// Mitsubishi GX Works2 project: q02 최종   PLC: Q02/Q02H

PROGRAM MAIN
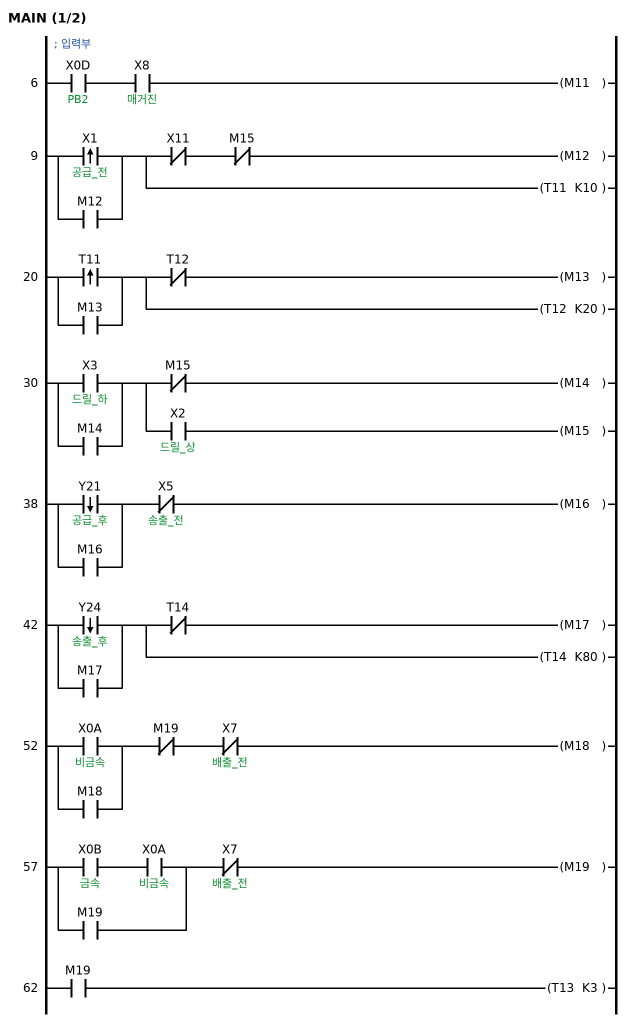
; 입력부
6     LD      X0D  ; PB2
      AND     X8  ; 매거진
      OUT     M11
9     LDP     X1  ; 공급_전
      OR      M12
      MPS
      ANI     X11
      ANI     M15
      OUT     M12
      MPP
      OUT     T11 K10
20    LDP     T11
      OR      M13
      MPS
      ANI     T12
      OUT     M13
      MPP
      OUT     T12 K20
30    LD      X3  ; 드릴_하
      OR      M14
      MPS
      ANI     M15
      OUT     M14
      MPP
      AND     X2  ; 드릴_상
      OUT     M15
38    LDF     Y21  ; 공급_후
      OR      M16
      ANI     X5  ; 송출_전
      OUT     M16
42    LDF     Y24  ; 송출_후
      OR      M17
      MPS
      ANI     T14
      OUT     M17
      MPP
      OUT     T14 K80
52    LD      X0A  ; 비금속
      OR      M18
      ANI     M19
      ANI     X7  ; 배출_전
      OUT     M18
57    LD      X0B  ; 금속
      AND     X0A  ; 비금속
      OR      M19
      ANI     X7  ; 배출_전
      OUT     M19
62    LD      M19
      OUT     T13 K3
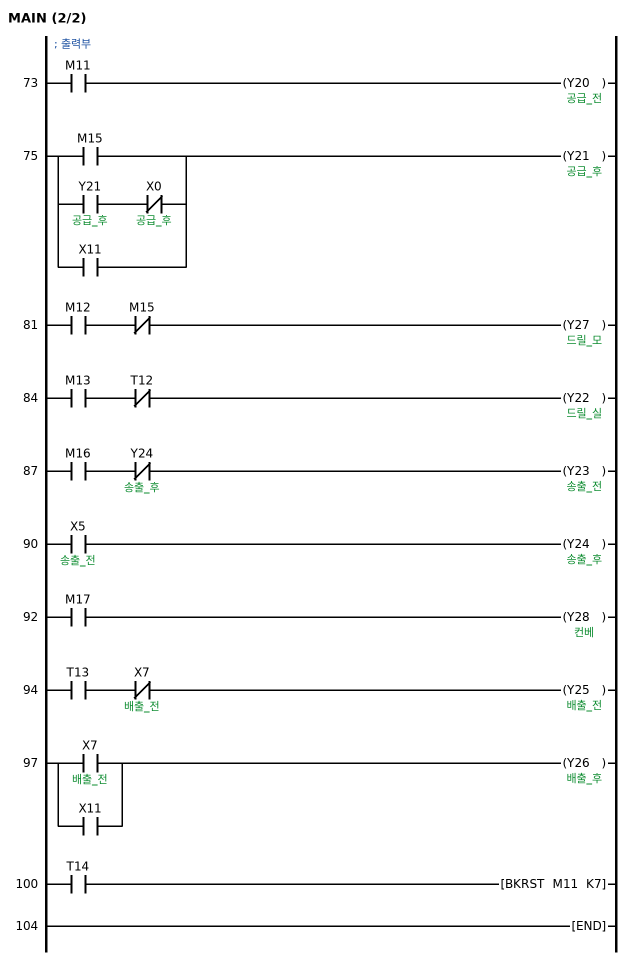
; 출력부
73    LD      M11
      OUT     Y20  ; 공급_전
75    LD      M15
      LD      Y21  ; 공급_후
      ANI     X0  ; 공급_후
      ORB
      OR      X11
      OUT     Y21  ; 공급_후
81    LD      M12
      ANI     M15
      OUT     Y27  ; 드릴_모
84    LD      M13
      ANI     T12
      OUT     Y22  ; 드릴_실
87    LD      M16
      ANI     Y24  ; 송출_후
      OUT     Y23  ; 송출_전
90    LD      X5  ; 송출_전
      OUT     Y24  ; 송출_후
92    LD      M17
      OUT     Y28  ; 컨베
94    LD      T13
      ANI     X7  ; 배출_전
      OUT     Y25  ; 배출_전
97    LD      X7  ; 배출_전
      OR      X11
      OUT     Y26  ; 배출_후
100   LD      T14
      BKRST   M11 K7
104   END
END_PROGRAM

// device comments not shown above
X4  ; 송출_후
X6  ; 배출_후
X9  ; 이송감지
X0C  ; PB1
X0E  ; PB3
X0F  ; 비상정지
Y29  ; 적램
Y2A  ; 황램
Y2B  ; 녹램
